// TIA Portal V17 export
// export: Created 2024-08-20T17:21:09.0209647Z, ExportSetting WithDefaults, DisplayName Totally Integrated Automation Portal, DisplayVersion V17 Update 4, DisplayName TIA Portal Openness, DisplayVersion V17 Update 4, DisplayName TIA Portal Version Control Interface, DisplayVersion V17, DisplayName STEP 7 Professional, DisplayVersion V17 Update 4, DisplayName STEP 7 Safety, DisplayVersion V17, DisplayName WinCC Advanced, DisplayVersion V17 Update 4
ORGANIZATION_BLOCK "CYC_INT5"   // OB35, LAD, CyclicInterrupt
TITLE = CONTROLE DE PID
{ S7_Optimized_Access := 'FALSE' }
VERSION : 0.1
// stored: AutoNumber false, IsIECCheckEnabled false, SetENOAutomatically false
   VAR_TEMP
      OB35_EV_CLASS : Byte;
      OB35_STRT_INF : Byte;
      OB35_PRIORITY : Byte;
      OB35_OB_NUMBR : Byte;
      OB35_RESERVED_1 : Byte;
      OB35_RESERVED_2 : Byte;
      OB35_PHASE_OFFSET : Word;
      OB35_RESERVED_3 : Int;
      OB35_EXC_FREQ : Int;
      OB35_DATE_TIME : Date_And_Time;
      "SPM-EEEB" : Real;   // Setpoint manual PID tanque de aeração 1
      EEEB_IT : Time;   // Ajuste integral do PID
      EEEB_DT : Time;   // Ajuste derivativo do PID
      EEEB_AUX : Real;   // Setpoint manual PID - auxiliar
      EEEB_P : Real;   // Setpoint manual PID - auxiliar
   END_VAR
   VAR_TEMP   // added for the SCL form of the ladder/FBD networks
      _w1 : Bool;
      _w2 : Bool;
      _w3 : Bool;
      _w4 : Bool;
   END_VAR
BEGIN

NETWORK
TITLE = CONVERSÃO DOS SETPOINTS PARA TEMPO PID EEEB


//CONVERSÃO DOS SETPOINTS DE TEMPO PID EEEB
      L     "PID"."PID-EEEB-I";
      L     1000.0;
      *R;
      RND;
      T     #EEEB_IT;

      L     "PID"."PID-EEEB-D";
      L     1000.0;
      *R;
      RND;
      T     #EEEB_DT;

      L     "PID"."PID-EEEB-P";
      L     -1.0;
      *R;
      T     #EEEB_P;


REGION Network 2: PID TANQUE DE AERAÇÃO 1
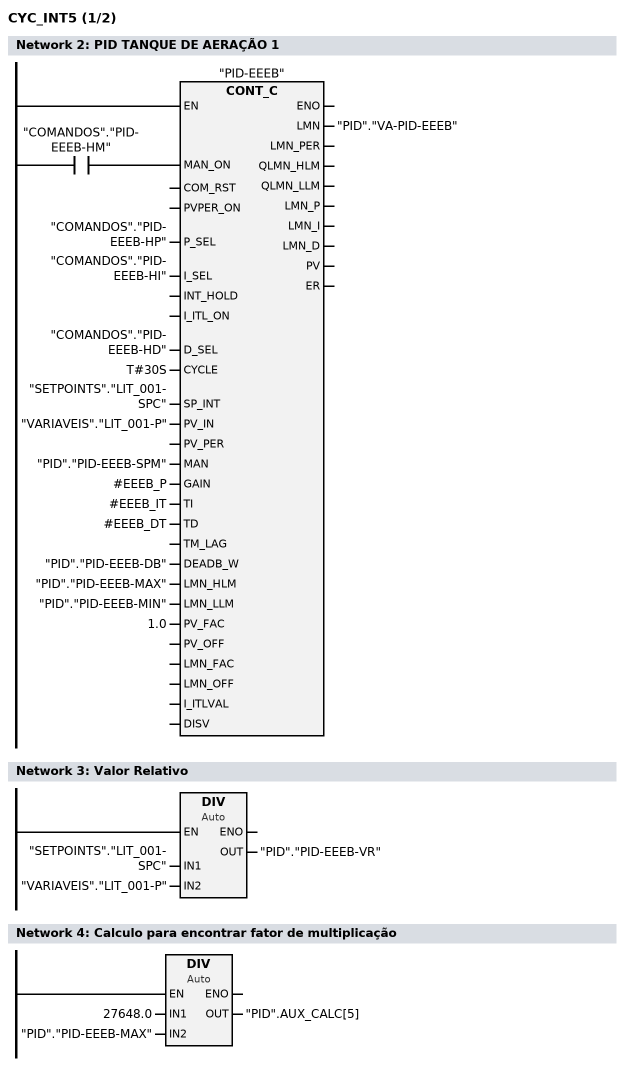
   RUNG wire#powerrail
      "PID-EEEB".CONT_C(MAN_ON := wire#w1, COM_RST :=, PVPER_ON :=, P_SEL := "COMANDOS"."PID-EEEB-HP", I_SEL := "COMANDOS"."PID-EEEB-HI", INT_HOLD :=, I_ITL_ON :=, D_SEL := "COMANDOS"."PID-EEEB-HD", CYCLE := T#30S, SP_INT := "SETPOINTS"."LIT_001-SPC", PV_IN := "VARIAVEIS"."LIT_001-P", PV_PER :=, MAN := "PID"."PID-EEEB-SPM", GAIN := #EEEB_P, TI := #EEEB_IT, TD := #EEEB_DT, TM_LAG :=, DEADB_W := "PID"."PID-EEEB-DB", LMN_HLM := "PID"."PID-EEEB-MAX", LMN_LLM := "PID"."PID-EEEB-MIN", PV_FAC := 1.0, PV_OFF :=, LMN_FAC :=, LMN_OFF :=, I_ITLVAL :=, DISV :=, LMN => "PID"."VA-PID-EEEB", LMN_PER =>, QLMN_HLM =>, QLMN_LLM =>, LMN_P =>, LMN_I =>, LMN_D =>, PV =>, ER =>)
   END_RUNG
   RUNG wire#powerrail
      Contact( "COMANDOS"."PID-EEEB-HM" )
   END_RUNG wire#w1
   // the same network as SCL:
   "PID-EEEB"(MAN_ON := "COMANDOS"."PID-EEEB-HM",   // CONT_C
              P_SEL := "COMANDOS"."PID-EEEB-HP",
              I_SEL := "COMANDOS"."PID-EEEB-HI",
              D_SEL := "COMANDOS"."PID-EEEB-HD",
              CYCLE := T#30S,
              SP_INT := "SETPOINTS"."LIT_001-SPC",
              PV_IN := "VARIAVEIS"."LIT_001-P",
              MAN := "PID"."PID-EEEB-SPM",
              GAIN := #EEEB_P,
              TI := #EEEB_IT,
              TD := #EEEB_DT,
              DEADB_W := "PID"."PID-EEEB-DB",
              LMN_HLM := "PID"."PID-EEEB-MAX",
              LMN_LLM := "PID"."PID-EEEB-MIN",
              PV_FAC := 1.0,
              LMN => "PID"."VA-PID-EEEB");
END_REGION

REGION Network 3: Valor Relativo
   RUNG wire#powerrail
      Div(in1 := "SETPOINTS"."LIT_001-SPC", in2 := "VARIAVEIS"."LIT_001-P", out => "PID"."PID-EEEB-VR")
   END_RUNG
   // the same network as SCL:
   "PID"."PID-EEEB-VR" := "SETPOINTS"."LIT_001-SPC" / "VARIAVEIS"."LIT_001-P";
END_REGION

REGION Network 4: Calculo para encontrar fator de multiplicação
   RUNG wire#powerrail
      Div(in1 := 27648.0, in2 := "PID"."PID-EEEB-MAX", out => "PID".AUX_CALC[5])
   END_RUNG
   // the same network as SCL:
   "PID".AUX_CALC[5] := 27648.0 / "PID"."PID-EEEB-MAX";
END_REGION

REGION Network 5: Movimenta saida PID para entrada analógica inversor
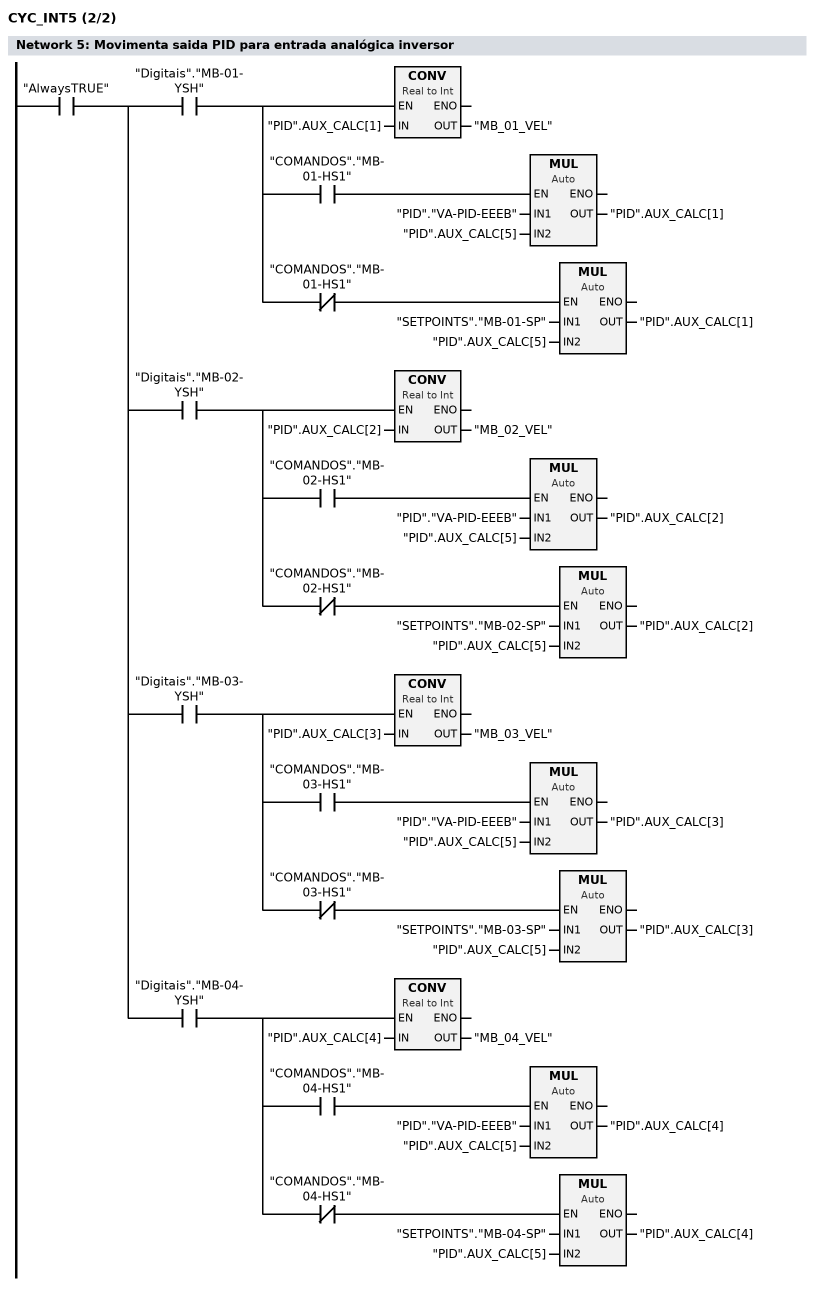
   RUNG wire#powerrail
      Contact( "AlwaysTRUE" )
      wire#w1
      Contact( "Digitais"."MB-01-YSH" )
      wire#w2
      { S7_Templates := "[SrcType := Real, DestType := Int]" } Convert(in := "PID".AUX_CALC[1], out => "MB_01_VEL")
   END_RUNG
   RUNG wire#w2
      Contact( "COMANDOS"."MB-01-HS1" )
      Mul(in1 := "PID"."VA-PID-EEEB", in2 := "PID".AUX_CALC[5], out => "PID".AUX_CALC[1])
   END_RUNG
   RUNG wire#w2
      I_Contact( "COMANDOS"."MB-01-HS1" )
      Mul(in1 := "SETPOINTS"."MB-01-SP", in2 := "PID".AUX_CALC[5], out => "PID".AUX_CALC[1])
   END_RUNG
   RUNG wire#w1
      Contact( "Digitais"."MB-02-YSH" )
      wire#w3
      { S7_Templates := "[SrcType := Real, DestType := Int]" } Convert(in := "PID".AUX_CALC[2], out => "MB_02_VEL")
   END_RUNG
   RUNG wire#w3
      Contact( "COMANDOS"."MB-02-HS1" )
      Mul(in1 := "PID"."VA-PID-EEEB", in2 := "PID".AUX_CALC[5], out => "PID".AUX_CALC[2])
   END_RUNG
   RUNG wire#w3
      I_Contact( "COMANDOS"."MB-02-HS1" )
      Mul(in1 := "SETPOINTS"."MB-02-SP", in2 := "PID".AUX_CALC[5], out => "PID".AUX_CALC[2])
   END_RUNG
   RUNG wire#w1
      Contact( "Digitais"."MB-03-YSH" )
      wire#w4
      { S7_Templates := "[SrcType := Real, DestType := Int]" } Convert(in := "PID".AUX_CALC[3], out => "MB_03_VEL")
   END_RUNG
   RUNG wire#w4
      Contact( "COMANDOS"."MB-03-HS1" )
      Mul(in1 := "PID"."VA-PID-EEEB", in2 := "PID".AUX_CALC[5], out => "PID".AUX_CALC[3])
   END_RUNG
   RUNG wire#w4
      I_Contact( "COMANDOS"."MB-03-HS1" )
      Mul(in1 := "SETPOINTS"."MB-03-SP", in2 := "PID".AUX_CALC[5], out => "PID".AUX_CALC[3])
   END_RUNG
   RUNG wire#w1
      Contact( "Digitais"."MB-04-YSH" )
      wire#w5
      { S7_Templates := "[SrcType := Real, DestType := Int]" } Convert(in := "PID".AUX_CALC[4], out => "MB_04_VEL")
   END_RUNG
   RUNG wire#w5
      Contact( "COMANDOS"."MB-04-HS1" )
      Mul(in1 := "PID"."VA-PID-EEEB", in2 := "PID".AUX_CALC[5], out => "PID".AUX_CALC[4])
   END_RUNG
   RUNG wire#w5
      I_Contact( "COMANDOS"."MB-04-HS1" )
      Mul(in1 := "SETPOINTS"."MB-04-SP", in2 := "PID".AUX_CALC[5], out => "PID".AUX_CALC[4])
   END_RUNG
   // the same network as SCL:
   #_w1 := "AlwaysTRUE" AND "Digitais"."MB-01-YSH";
   IF #_w1 THEN "MB_01_VEL" := REAL_TO_INT("PID".AUX_CALC[1]); END_IF;
   IF #_w1 AND "COMANDOS"."MB-01-HS1" THEN
       "PID".AUX_CALC[1] := "PID"."VA-PID-EEEB" * "PID".AUX_CALC[5];
   END_IF;
   IF #_w1 AND NOT "COMANDOS"."MB-01-HS1" THEN
       "PID".AUX_CALC[1] := "SETPOINTS"."MB-01-SP" * "PID".AUX_CALC[5];
   END_IF;
   #_w2 := "AlwaysTRUE" AND "Digitais"."MB-02-YSH";
   IF #_w2 THEN "MB_02_VEL" := REAL_TO_INT("PID".AUX_CALC[2]); END_IF;
   IF #_w2 AND "COMANDOS"."MB-02-HS1" THEN
       "PID".AUX_CALC[2] := "PID"."VA-PID-EEEB" * "PID".AUX_CALC[5];
   END_IF;
   IF #_w2 AND NOT "COMANDOS"."MB-02-HS1" THEN
       "PID".AUX_CALC[2] := "SETPOINTS"."MB-02-SP" * "PID".AUX_CALC[5];
   END_IF;
   #_w3 := "AlwaysTRUE" AND "Digitais"."MB-03-YSH";
   IF #_w3 THEN "MB_03_VEL" := REAL_TO_INT("PID".AUX_CALC[3]); END_IF;
   IF #_w3 AND "COMANDOS"."MB-03-HS1" THEN
       "PID".AUX_CALC[3] := "PID"."VA-PID-EEEB" * "PID".AUX_CALC[5];
   END_IF;
   IF #_w3 AND NOT "COMANDOS"."MB-03-HS1" THEN
       "PID".AUX_CALC[3] := "SETPOINTS"."MB-03-SP" * "PID".AUX_CALC[5];
   END_IF;
   #_w4 := "AlwaysTRUE" AND "Digitais"."MB-04-YSH";
   IF #_w4 THEN "MB_04_VEL" := REAL_TO_INT("PID".AUX_CALC[4]); END_IF;
   IF #_w4 AND "COMANDOS"."MB-04-HS1" THEN
       "PID".AUX_CALC[4] := "PID"."VA-PID-EEEB" * "PID".AUX_CALC[5];
   END_IF;
   IF #_w4 AND NOT "COMANDOS"."MB-04-HS1" THEN
       "PID".AUX_CALC[4] := "SETPOINTS"."MB-04-SP" * "PID".AUX_CALC[5];
   END_IF;
END_REGION
END_ORGANIZATION_BLOCK
